// TIA Portal V17 export
// export: Created 2023-05-12T10:40:25.6107869Z, DisplayName Totally Integrated Automation Portal, DisplayVersion V17 Update 4, DisplayName TIA Portal Openness, DisplayVersion V17 Update 4, DisplayName TIA Portal Version Control Interface, DisplayVersion V17, DisplayName STEP 7 Professional, DisplayVersion V17 Update 4, DisplayName STEP 7 Safety, DisplayVersion V17, DisplayName WinCC Advanced / Unified PC, DisplayVersion V17 Update 4
FUNCTION_BLOCK "FB_EM_InputConditioning"   // FB19, LAD
{ S7_Optimized_Access := 'TRUE' }
VERSION : 0.1
// stored: AutoNumber true, CodeModifiedDate 2023-05-12T12:59:41.6492354Z, CompileDate 2023-05-12T12:59:41.6492354Z, CreationDate 2023-05-08T12:19:11.3376827Z, DownloadWithoutReinit false, HandleErrorsWithinBlock false, InterfaceModifiedDate 2023-05-12T12:59:19.7337351Z, IsConsistent true, IsIECCheckEnabled false, IsKnowHowProtected false, IsRetainMemResEnabled false, IsWriteProtected false, LibraryConformanceStatus Warning: The object contains access to global data blocks., MemoryReserve 100, ModifiedDate 2023-05-12T12:59:41.6492354Z, ParameterModified 2022-09-13T10:25:33.4387708Z, PLCSimAdvancedSupport true, SetENOAutomatically false, StructureModified 2023-05-12T12:59:19.7337351Z, UDAEnableTagReadback false
   VAR
      TT01_TempZasil_EC_Inst { S7_SetPoint := 'True'} : "FB_CM_MeasurementPoint";
      TT02_TempPowr_EC_Inst { S7_SetPoint := 'True'} : "FB_CM_MeasurementPoint";
      TT04_TempPowr_PLD3_Inst { S7_SetPoint := 'True'} : "FB_CM_MeasurementPoint";
      TT06_TempPowr_PLN3_Inst { S7_SetPoint := 'True'} : "FB_CM_MeasurementPoint";
      PT01_CisnZasil_EC_Inst { S7_SetPoint := 'True'} : "FB_CM_MeasurementPoint";
      PT02_CisnPowr_EC_Inst { S7_SetPoint := 'True'} : "FB_CM_MeasurementPoint";
      PT03_CisnZasil_PLD3_Inst { S7_SetPoint := 'True'} : "FB_CM_MeasurementPoint";
      PT04_CisnPowr_PLD3_Inst { S7_SetPoint := 'True'} : "FB_CM_MeasurementPoint";
      PT05_CisnZasil_PLN3_Inst { S7_SetPoint := 'True'} : "FB_CM_MeasurementPoint";
      PT06_CisnPowr_PLN3_Inst { S7_SetPoint := 'True'} : "FB_CM_MeasurementPoint";
      TTs_TempSzafy_Inst { S7_SetPoint := 'True'} : "FB_CM_MeasurementPoint";
      TTk_TempKom_Inst { S7_SetPoint := 'True'} : "FB_CM_MeasurementPoint";
   END_VAR
BEGIN

REGION Network 1: TT01_TempZasil_EC - Temperatura zasilania z EC
   // TT01_TempZasil_EC - Temperatura zasilania z EC
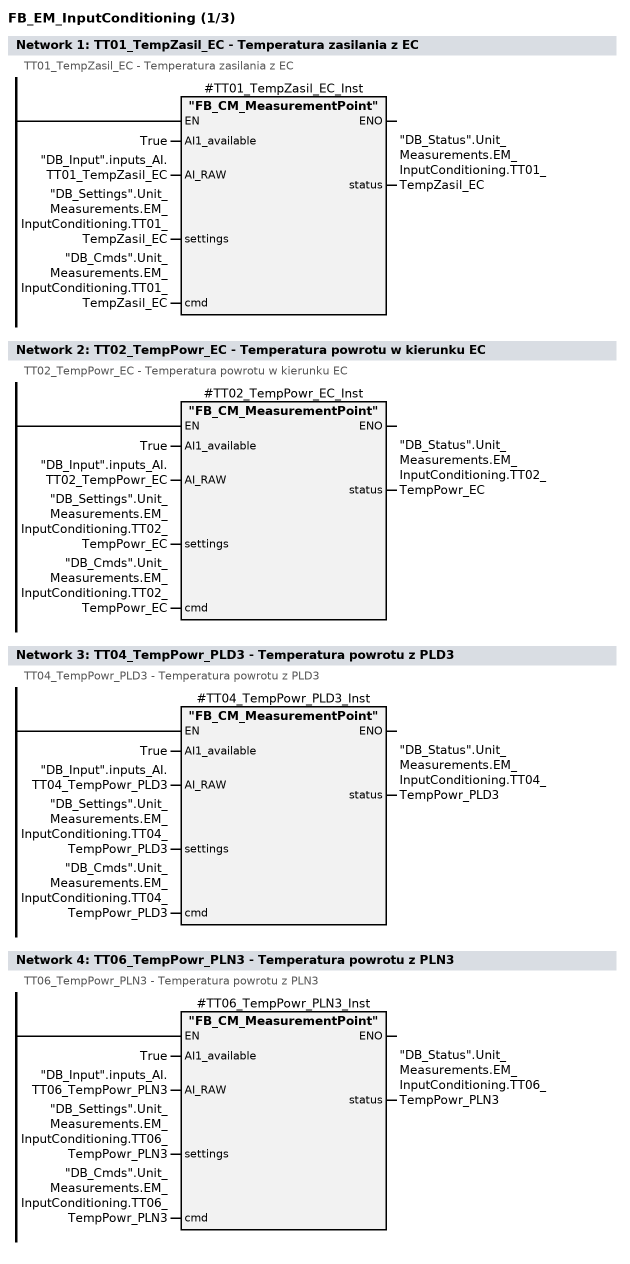
   RUNG wire#powerrail
      #TT01_TempZasil_EC_Inst(AI1_available := True, AI_RAW := "DB_Input".inputs_AI.TT01_TempZasil_EC, settings := "DB_Settings".Unit_Measurements.EM_InputConditioning.TT01_TempZasil_EC, cmd := "DB_Cmds".Unit_Measurements.EM_InputConditioning.TT01_TempZasil_EC, status => "DB_Status".Unit_Measurements.EM_InputConditioning.TT01_TempZasil_EC)
   END_RUNG
   // the same network as SCL:
   #TT01_TempZasil_EC_Inst(AI1_available := True,   // "FB_CM_MeasurementPoint"
                           AI_RAW := "DB_Input".inputs_AI.TT01_TempZasil_EC,
                           settings := "DB_Settings".Unit_Measurements.EM_InputConditioning.TT01_TempZasil_EC,
                           cmd := "DB_Cmds".Unit_Measurements.EM_InputConditioning.TT01_TempZasil_EC,
                           status => "DB_Status".Unit_Measurements.EM_InputConditioning.TT01_TempZasil_EC);
END_REGION

REGION Network 2: TT02_TempPowr_EC - Temperatura powrotu w kierunku EC
   // TT02_TempPowr_EC - Temperatura powrotu w kierunku EC
   RUNG wire#powerrail
      #TT02_TempPowr_EC_Inst(AI1_available := True, AI_RAW := "DB_Input".inputs_AI.TT02_TempPowr_EC, settings := "DB_Settings".Unit_Measurements.EM_InputConditioning.TT02_TempPowr_EC, cmd := "DB_Cmds".Unit_Measurements.EM_InputConditioning.TT02_TempPowr_EC, status => "DB_Status".Unit_Measurements.EM_InputConditioning.TT02_TempPowr_EC)
   END_RUNG
   // the same network as SCL:
   #TT02_TempPowr_EC_Inst(AI1_available := True,   // "FB_CM_MeasurementPoint"
                          AI_RAW := "DB_Input".inputs_AI.TT02_TempPowr_EC,
                          settings := "DB_Settings".Unit_Measurements.EM_InputConditioning.TT02_TempPowr_EC,
                          cmd := "DB_Cmds".Unit_Measurements.EM_InputConditioning.TT02_TempPowr_EC,
                          status => "DB_Status".Unit_Measurements.EM_InputConditioning.TT02_TempPowr_EC);
END_REGION

REGION Network 3: TT04_TempPowr_PLD3 - Temperatura powrotu z PLD3
   // TT04_TempPowr_PLD3 - Temperatura powrotu z PLD3
   RUNG wire#powerrail
      #TT04_TempPowr_PLD3_Inst(AI1_available := True, AI_RAW := "DB_Input".inputs_AI.TT04_TempPowr_PLD3, settings := "DB_Settings".Unit_Measurements.EM_InputConditioning.TT04_TempPowr_PLD3, cmd := "DB_Cmds".Unit_Measurements.EM_InputConditioning.TT04_TempPowr_PLD3, status => "DB_Status".Unit_Measurements.EM_InputConditioning.TT04_TempPowr_PLD3)
   END_RUNG
   // the same network as SCL:
   #TT04_TempPowr_PLD3_Inst(AI1_available := True,   // "FB_CM_MeasurementPoint"
                           AI_RAW := "DB_Input".inputs_AI.TT04_TempPowr_PLD3,
                           settings := "DB_Settings".Unit_Measurements.EM_InputConditioning.TT04_TempPowr_PLD3,
                           cmd := "DB_Cmds".Unit_Measurements.EM_InputConditioning.TT04_TempPowr_PLD3,
                           status => "DB_Status".Unit_Measurements.EM_InputConditioning.TT04_TempPowr_PLD3);
END_REGION

REGION Network 4: TT06_TempPowr_PLN3 - Temperatura powrotu z PLN3
   // TT06_TempPowr_PLN3 - Temperatura powrotu z PLN3
   RUNG wire#powerrail
      #TT06_TempPowr_PLN3_Inst(AI1_available := True, AI_RAW := "DB_Input".inputs_AI.TT06_TempPowr_PLN3, settings := "DB_Settings".Unit_Measurements.EM_InputConditioning.TT06_TempPowr_PLN3, cmd := "DB_Cmds".Unit_Measurements.EM_InputConditioning.TT06_TempPowr_PLN3, status => "DB_Status".Unit_Measurements.EM_InputConditioning.TT06_TempPowr_PLN3)
   END_RUNG
   // the same network as SCL:
   #TT06_TempPowr_PLN3_Inst(AI1_available := True,   // "FB_CM_MeasurementPoint"
                           AI_RAW := "DB_Input".inputs_AI.TT06_TempPowr_PLN3,
                           settings := "DB_Settings".Unit_Measurements.EM_InputConditioning.TT06_TempPowr_PLN3,
                           cmd := "DB_Cmds".Unit_Measurements.EM_InputConditioning.TT06_TempPowr_PLN3,
                           status => "DB_Status".Unit_Measurements.EM_InputConditioning.TT06_TempPowr_PLN3);
END_REGION

REGION Network 5: PT01_CisnZasil_EC - CIśnienie zasilania z EC
   // PT01_CisnZasil_EC - CIśnienie zasilania z EC
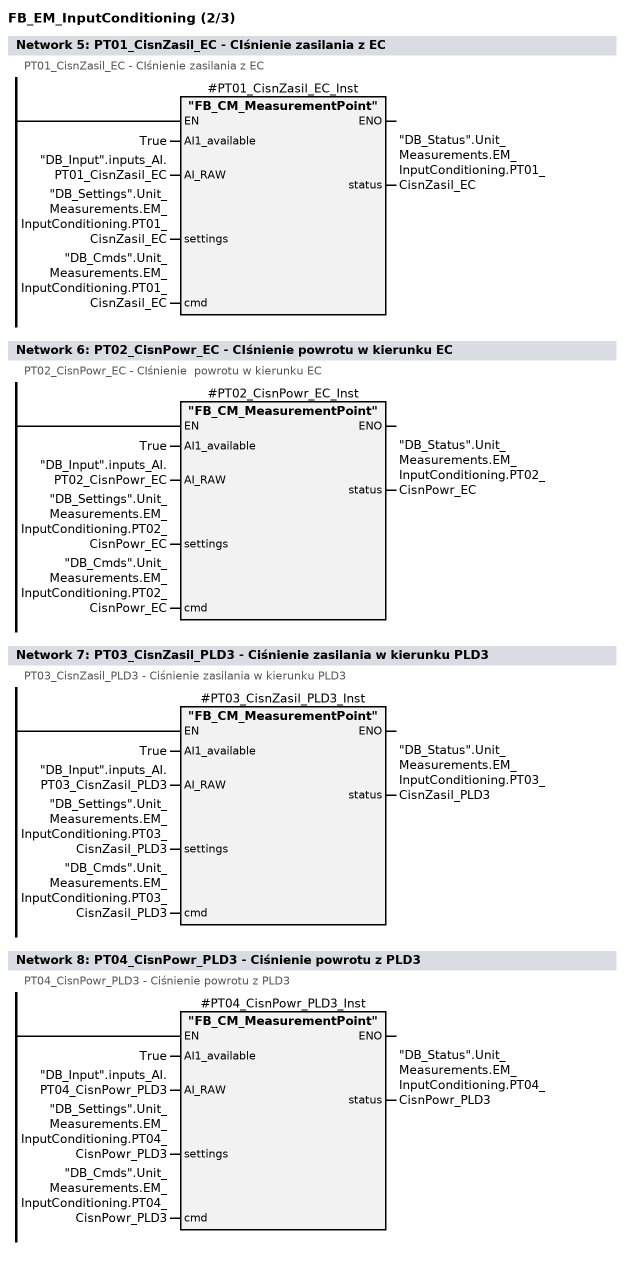
   RUNG wire#powerrail
      #PT01_CisnZasil_EC_Inst(AI1_available := True, AI_RAW := "DB_Input".inputs_AI.PT01_CisnZasil_EC, settings := "DB_Settings".Unit_Measurements.EM_InputConditioning.PT01_CisnZasil_EC, cmd := "DB_Cmds".Unit_Measurements.EM_InputConditioning.PT01_CisnZasil_EC, status => "DB_Status".Unit_Measurements.EM_InputConditioning.PT01_CisnZasil_EC)
   END_RUNG
   // the same network as SCL:
   #PT01_CisnZasil_EC_Inst(AI1_available := True,   // "FB_CM_MeasurementPoint"
                           AI_RAW := "DB_Input".inputs_AI.PT01_CisnZasil_EC,
                           settings := "DB_Settings".Unit_Measurements.EM_InputConditioning.PT01_CisnZasil_EC,
                           cmd := "DB_Cmds".Unit_Measurements.EM_InputConditioning.PT01_CisnZasil_EC,
                           status => "DB_Status".Unit_Measurements.EM_InputConditioning.PT01_CisnZasil_EC);
END_REGION

REGION Network 6: PT02_CisnPowr_EC - CIśnienie powrotu w kierunku EC
   // PT02_CisnPowr_EC - CIśnienie  powrotu w kierunku EC
   RUNG wire#powerrail
      #PT02_CisnPowr_EC_Inst(AI1_available := True, AI_RAW := "DB_Input".inputs_AI.PT02_CisnPowr_EC, settings := "DB_Settings".Unit_Measurements.EM_InputConditioning.PT02_CisnPowr_EC, cmd := "DB_Cmds".Unit_Measurements.EM_InputConditioning.PT02_CisnPowr_EC, status => "DB_Status".Unit_Measurements.EM_InputConditioning.PT02_CisnPowr_EC)
   END_RUNG
   // the same network as SCL:
   #PT02_CisnPowr_EC_Inst(AI1_available := True,   // "FB_CM_MeasurementPoint"
                          AI_RAW := "DB_Input".inputs_AI.PT02_CisnPowr_EC,
                          settings := "DB_Settings".Unit_Measurements.EM_InputConditioning.PT02_CisnPowr_EC,
                          cmd := "DB_Cmds".Unit_Measurements.EM_InputConditioning.PT02_CisnPowr_EC,
                          status => "DB_Status".Unit_Measurements.EM_InputConditioning.PT02_CisnPowr_EC);
END_REGION

REGION Network 7: PT03_CisnZasil_PLD3 - Ciśnienie zasilania w kierunku PLD3
   // PT03_CisnZasil_PLD3 - Ciśnienie zasilania w kierunku PLD3
   RUNG wire#powerrail
      #PT03_CisnZasil_PLD3_Inst(AI1_available := True, AI_RAW := "DB_Input".inputs_AI.PT03_CisnZasil_PLD3, settings := "DB_Settings".Unit_Measurements.EM_InputConditioning.PT03_CisnZasil_PLD3, cmd := "DB_Cmds".Unit_Measurements.EM_InputConditioning.PT03_CisnZasil_PLD3, status => "DB_Status".Unit_Measurements.EM_InputConditioning.PT03_CisnZasil_PLD3)
   END_RUNG
   // the same network as SCL:
   #PT03_CisnZasil_PLD3_Inst(AI1_available := True,   // "FB_CM_MeasurementPoint"
                           AI_RAW := "DB_Input".inputs_AI.PT03_CisnZasil_PLD3,
                           settings := "DB_Settings".Unit_Measurements.EM_InputConditioning.PT03_CisnZasil_PLD3,
                           cmd := "DB_Cmds".Unit_Measurements.EM_InputConditioning.PT03_CisnZasil_PLD3,
                           status => "DB_Status".Unit_Measurements.EM_InputConditioning.PT03_CisnZasil_PLD3);
END_REGION

REGION Network 8: PT04_CisnPowr_PLD3 - Ciśnienie powrotu z PLD3
   // PT04_CisnPowr_PLD3 - Ciśnienie powrotu z PLD3
   RUNG wire#powerrail
      #PT04_CisnPowr_PLD3_Inst(AI1_available := True, AI_RAW := "DB_Input".inputs_AI.PT04_CisnPowr_PLD3, settings := "DB_Settings".Unit_Measurements.EM_InputConditioning.PT04_CisnPowr_PLD3, cmd := "DB_Cmds".Unit_Measurements.EM_InputConditioning.PT04_CisnPowr_PLD3, status => "DB_Status".Unit_Measurements.EM_InputConditioning.PT04_CisnPowr_PLD3)
   END_RUNG
   // the same network as SCL:
   #PT04_CisnPowr_PLD3_Inst(AI1_available := True,   // "FB_CM_MeasurementPoint"
                           AI_RAW := "DB_Input".inputs_AI.PT04_CisnPowr_PLD3,
                           settings := "DB_Settings".Unit_Measurements.EM_InputConditioning.PT04_CisnPowr_PLD3,
                           cmd := "DB_Cmds".Unit_Measurements.EM_InputConditioning.PT04_CisnPowr_PLD3,
                           status => "DB_Status".Unit_Measurements.EM_InputConditioning.PT04_CisnPowr_PLD3);
END_REGION

REGION Network 9: PT05_CisnZasil_PLN3 - Ciśnienie zasilania w kierunku PLN3
   // PT05_CisnZasil_PLN3 - Ciśnienie zasilania w kierunku PLN3
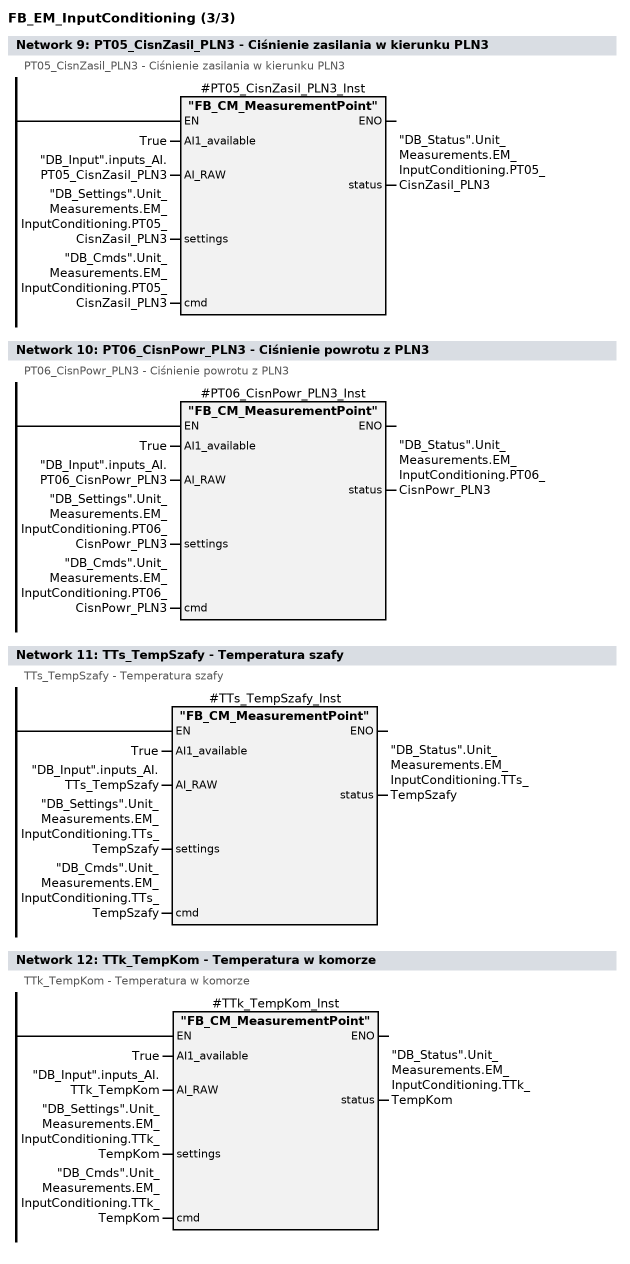
   RUNG wire#powerrail
      #PT05_CisnZasil_PLN3_Inst(AI1_available := True, AI_RAW := "DB_Input".inputs_AI.PT05_CisnZasil_PLN3, settings := "DB_Settings".Unit_Measurements.EM_InputConditioning.PT05_CisnZasil_PLN3, cmd := "DB_Cmds".Unit_Measurements.EM_InputConditioning.PT05_CisnZasil_PLN3, status => "DB_Status".Unit_Measurements.EM_InputConditioning.PT05_CisnZasil_PLN3)
   END_RUNG
   // the same network as SCL:
   #PT05_CisnZasil_PLN3_Inst(AI1_available := True,   // "FB_CM_MeasurementPoint"
                           AI_RAW := "DB_Input".inputs_AI.PT05_CisnZasil_PLN3,
                           settings := "DB_Settings".Unit_Measurements.EM_InputConditioning.PT05_CisnZasil_PLN3,
                           cmd := "DB_Cmds".Unit_Measurements.EM_InputConditioning.PT05_CisnZasil_PLN3,
                           status => "DB_Status".Unit_Measurements.EM_InputConditioning.PT05_CisnZasil_PLN3);
END_REGION

REGION Network 10: PT06_CisnPowr_PLN3 - Ciśnienie powrotu z PLN3
   // PT06_CisnPowr_PLN3 - Ciśnienie powrotu z PLN3
   RUNG wire#powerrail
      #PT06_CisnPowr_PLN3_Inst(AI1_available := True, AI_RAW := "DB_Input".inputs_AI.PT06_CisnPowr_PLN3, settings := "DB_Settings".Unit_Measurements.EM_InputConditioning.PT06_CisnPowr_PLN3, cmd := "DB_Cmds".Unit_Measurements.EM_InputConditioning.PT06_CisnPowr_PLN3, status => "DB_Status".Unit_Measurements.EM_InputConditioning.PT06_CisnPowr_PLN3)
   END_RUNG
   // the same network as SCL:
   #PT06_CisnPowr_PLN3_Inst(AI1_available := True,   // "FB_CM_MeasurementPoint"
                           AI_RAW := "DB_Input".inputs_AI.PT06_CisnPowr_PLN3,
                           settings := "DB_Settings".Unit_Measurements.EM_InputConditioning.PT06_CisnPowr_PLN3,
                           cmd := "DB_Cmds".Unit_Measurements.EM_InputConditioning.PT06_CisnPowr_PLN3,
                           status => "DB_Status".Unit_Measurements.EM_InputConditioning.PT06_CisnPowr_PLN3);
END_REGION

REGION Network 11: TTs_TempSzafy - Temperatura szafy
   // TTs_TempSzafy - Temperatura szafy
   RUNG wire#powerrail
      #TTs_TempSzafy_Inst(AI1_available := True, AI_RAW := "DB_Input".inputs_AI.TTs_TempSzafy, settings := "DB_Settings".Unit_Measurements.EM_InputConditioning.TTs_TempSzafy, cmd := "DB_Cmds".Unit_Measurements.EM_InputConditioning.TTs_TempSzafy, status => "DB_Status".Unit_Measurements.EM_InputConditioning.TTs_TempSzafy)
   END_RUNG
   // the same network as SCL:
   #TTs_TempSzafy_Inst(AI1_available := True,   // "FB_CM_MeasurementPoint"
                       AI_RAW := "DB_Input".inputs_AI.TTs_TempSzafy,
                       settings := "DB_Settings".Unit_Measurements.EM_InputConditioning.TTs_TempSzafy,
                       cmd := "DB_Cmds".Unit_Measurements.EM_InputConditioning.TTs_TempSzafy,
                       status => "DB_Status".Unit_Measurements.EM_InputConditioning.TTs_TempSzafy);
END_REGION

REGION Network 12: TTk_TempKom - Temperatura w komorze
   // TTk_TempKom - Temperatura w komorze
   RUNG wire#powerrail
      #TTk_TempKom_Inst(AI1_available := True, AI_RAW := "DB_Input".inputs_AI.TTk_TempKom, settings := "DB_Settings".Unit_Measurements.EM_InputConditioning.TTk_TempKom, cmd := "DB_Cmds".Unit_Measurements.EM_InputConditioning.TTk_TempKom, status => "DB_Status".Unit_Measurements.EM_InputConditioning.TTk_TempKom)
   END_RUNG
   // the same network as SCL:
   #TTk_TempKom_Inst(AI1_available := True,   // "FB_CM_MeasurementPoint"
                     AI_RAW := "DB_Input".inputs_AI.TTk_TempKom,
                     settings := "DB_Settings".Unit_Measurements.EM_InputConditioning.TTk_TempKom,
                     cmd := "DB_Cmds".Unit_Measurements.EM_InputConditioning.TTk_TempKom,
                     status => "DB_Status".Unit_Measurements.EM_InputConditioning.TTk_TempKom);
END_REGION
END_FUNCTION_BLOCK
